Omron Sysmac Studio project Otopark_Uygulamasi (Sysmac Studio 1.65.0.64007, StandardProject)

# Controller new_Controller_0: NX1P2-1040DT1 version 1.69
Task PrimaryTask (priority 4, period or condition 2000): Program0

VAR_GLOBAL
    IN_Start_Buton : BOOL;
    IN_Stop_Buton : BOOL;
    IN_Giris_Sensoru : BOOL;
    IN_Cikis_Sensoru : BOOL;
    OUT_Giris_Bariyer_Ac : BOOL;
    OUT_Giris_Bariyer_Kapat : BOOL;
    OUT_Cikis_Bariyer_Ac : BOOL;
    OUT_Cikis_Bariyer_Kapat : BOOL;
    OUT_YesilLamba : BOOL;
    OUT_KirmiziLamba : BOOL;
END_VAR

PROGRAM Program0
VAR
    Start : BOOL;
    lale : TON;
    Arac_Kapasitesi : INT;
    Giris_Bariyeri_Acilmali : BOOL;
    TON_GirisBar1 : TON;
    Giris_Bariyeri_Acik : BOOL;
    TON_GirisBar2 : TON;
    Cikis_Bariyeri_Acilmali : BOOL;
    TON_CikisBar1 : TON;
    Cikis_Bariyeri_Acik : BOOL;
    TON_CikisBar2 : TON;
    INT<31 : INT;
END_VAR
VAR_EXTERNAL
    IN_Start_Buton : BOOL;
    IN_Stop_Buton : BOOL;
    IN_Giris_Sensoru : BOOL;
    OUT_Giris_Bariyer_Ac : BOOL;
    OUT_Giris_Bariyer_Kapat : BOOL;
    IN_Cikis_Sensoru : BOOL;
    OUT_Cikis_Bariyer_Ac : BOOL;
    OUT_Cikis_Bariyer_Kapat : BOOL;
    OUT_KirmiziLamba : BOOL;
    OUT_YesilLamba : BOOL;
END_VAR
VAR
    _e1 : R_TRIG;
    _p2 : BOOL;
    _e3 : R_TRIG;
    _p4 : BOOL;
    _e5 : R_TRIG;
END_VAR

(* Section Section0: ladder, written here as Structured Text *)

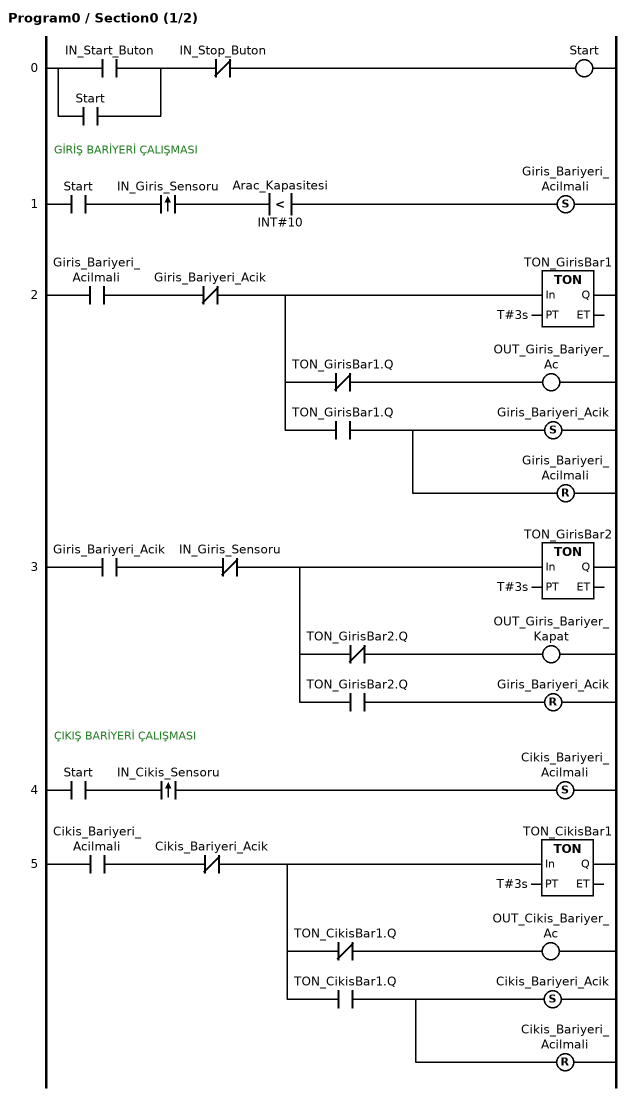
(* Rung 0 *)
Start := (IN_Start_Buton OR Start) AND NOT IN_Stop_Buton;
(* Rung 1: GİRİŞ BARİYERİ ÇALIŞMASI *)
_e1(CLK := IN_Giris_Sensoru);
IF Start AND _e1.Q AND (Arac_Kapasitesi < INT#10) THEN Giris_Bariyeri_Acilmali := TRUE; END_IF;
(* Rung 2 *)
_p2 := Giris_Bariyeri_Acilmali AND NOT Giris_Bariyeri_Acik;
TON_GirisBar1(In := _p2, PT := T#3s);
OUT_Giris_Bariyer_Ac := _p2 AND NOT TON_GirisBar1.Q;
IF _p2 AND TON_GirisBar1.Q THEN
    Giris_Bariyeri_Acik := TRUE;
    Giris_Bariyeri_Acilmali := FALSE;
END_IF;
(* Rung 3 *)
TON_GirisBar2(In := Giris_Bariyeri_Acik AND NOT IN_Giris_Sensoru, PT := T#3s);
OUT_Giris_Bariyer_Kapat := Giris_Bariyeri_Acik AND NOT IN_Giris_Sensoru AND NOT TON_GirisBar2.Q;
IF Giris_Bariyeri_Acik AND NOT IN_Giris_Sensoru AND TON_GirisBar2.Q THEN
    Giris_Bariyeri_Acik := FALSE;
END_IF;
(* Rung 4: ÇIKIŞ BARİYERİ ÇALIŞMASI *)
_e3(CLK := IN_Cikis_Sensoru);
IF Start AND _e3.Q THEN Cikis_Bariyeri_Acilmali := TRUE; END_IF;
(* Rung 5 *)
_p4 := Cikis_Bariyeri_Acilmali AND NOT Cikis_Bariyeri_Acik;
TON_CikisBar1(In := _p4, PT := T#3s);
OUT_Cikis_Bariyer_Ac := _p4 AND NOT TON_CikisBar1.Q;
IF _p4 AND TON_CikisBar1.Q THEN
    Cikis_Bariyeri_Acik := TRUE;
    Cikis_Bariyeri_Acilmali := FALSE;
END_IF;

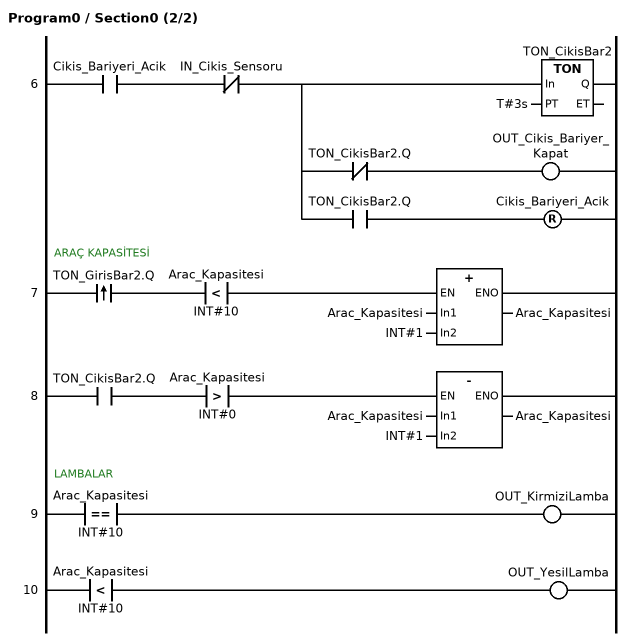
(* Rung 6 *)
TON_CikisBar2(In := Cikis_Bariyeri_Acik AND NOT IN_Cikis_Sensoru, PT := T#3s);
OUT_Cikis_Bariyer_Kapat := Cikis_Bariyeri_Acik AND NOT IN_Cikis_Sensoru AND NOT TON_CikisBar2.Q;
IF Cikis_Bariyeri_Acik AND NOT IN_Cikis_Sensoru AND TON_CikisBar2.Q THEN
    Cikis_Bariyeri_Acik := FALSE;
END_IF;
(* Rung 7: ARAÇ KAPASİTESİ *)
_e5(CLK := TON_GirisBar2.Q);
IF _e5.Q AND (Arac_Kapasitesi < INT#10) THEN Arac_Kapasitesi := Arac_Kapasitesi + INT#1; END_IF;
(* Rung 8 *)
IF TON_CikisBar2.Q AND (Arac_Kapasitesi > INT#0) THEN Arac_Kapasitesi := Arac_Kapasitesi - INT#1; END_IF;
(* Rung 9: LAMBALAR *)
OUT_KirmiziLamba := Arac_Kapasitesi = INT#10;
(* Rung 10 *)
OUT_YesilLamba := Arac_Kapasitesi < INT#10;
END_PROGRAM